(* IEC 61131-3 sources: std_i2980_v2.06_cp053/Source/IMM/ieccontrol/GlobalBaseArchives (part 5) *)

(* ---- FBStart.pu ---- *)
(*
IntermediateCond is optional(only needed for movements with intermediate conditions)
It starts from 1 to and goes up to the maximum intermediate condition
For movements without intermediate conditions it should be 0.

*)

IMPORT_OVER_LISTFILE
 SET_EVENT
, ASSERT
, tsDeviceId
, tMoveIdent
, tsMoveData
, tevStartData
, tevStart

END_IMPORT

FUNCTION_BLOCK FBStart #DUMMY_EDIT_BLOCK

VAR_INPUT
 DeviceId : tsDeviceId (* Device that should be started *);
 MoveDir : tMoveIdent (* Movement direction to start *);
 MoveId : tMoveIdent (* Movement ID to start *);
 IntermediateCond : DINT (* optional: Intermediate condition that should be used for the movement *);
 pbPosReached : REFTO BOOL (* optional: *);
 pMovementData : REFTO tsMoveData (* optional: Reference to the sv_MoveXxx *);
END_VAR

SYSTEM_VAR
 sv_bInitDone : BOOL;
END_VAR

SYSTEM_OBJECT
 evStart : tevStart;
 erAssert : ALARM;
END_OBJECT

VAR
 evStartData : tevStartData;
 dummy : BOOL;
END_VAR
#BEGIN_EDIT_BLOCK
(**************************************** WARNING ********************************************
 *** The KEBA Kemro K2 System including software is not intended for safety control tasks! ***
 ***                       For further information see Comment tab!                        ***
 *********************************************************************************************)

//if the movements are still not registered, gives application programmer code offset and frame offset
dummy := ASSERT(sv_bInitDone, erAssert);

//send start event
evStartData.DeviceId := DeviceId;
evStartData.MoveDir := MoveDir;
evStartData.MoveId := MoveId;
evStartData.IntermediateCond := IntermediateCond;
evStartData.pbPosReached := pbPosReached;
evStartData.pMovementData := pMovementData;
SET_EVENT(evStart,evStartData);

;#END_EDIT_BLOCK END_FUNCTION_BLOCK

#END_OF_IEC_PART

@Puma @IecEditor 6 96 @Pou 25
@@@BEG_Comment@@@
IntermediateCond is optional(only needed for movements with intermediate conditions)
It starts from 1 to and goes up to the maximum intermediate condition
For movements without intermediate conditions it should be 0.

@@@END_Comment@@@

@BEG_Contents

@BEG_Func
@RT(17)FuncTreeContainer
2
@Var @RT(9)SET_EVENT @RT(0) @T @T @DERIVED 0 @F @RT(23)KEBA_STANDARD_PROCEDURE @F
@T
@BEG_Attrib
0 @RT(0) @RT(0)
@END_Attrib
1 1 @F @F @F @F

@Var @RT(6)ASSERT @RT(0) @T @T @DERIVED 0 @F @RT(8)FUNCTION @F
@T
@BEG_Attrib
0 @RT(0) @RT(0)
@END_Attrib
1 1 @F @F @F @F

@END_Func

@BEG_Const
@RT(18)ConstTreeContainer
0
@END_Const

@BEG_Export

@BEG_Kind
@FUNCTION_BLOCK @RT(7)FBStart @STRUCTURED_TEXT
@RT(0) @RT(0) @RT(0)
@END_Kind

@BEG_Dcl
@RT(16)DclTreeContainer
11
@Var @RT(8)DeviceId @RT(0) @T @T @DERIVED 0 @T @T @DT @RT(10)tsDeviceId @RT(0) @T @T @UNKNOWN 0 @F
@F @F
@T
@BEG_Attrib
3 @RT(0) @RT(29)Device that should be started @RT(0)
@END_Attrib
1 1 @F @F @F @F

@Var @RT(7)MoveDir @RT(0) @T @T @DERIVED 0 @T @T @DT @RT(10)tMoveIdent @RT(0) @T @T @UNKNOWN 0 @F
@F @F
@T
@BEG_Attrib
3 @RT(0) @RT(27)Movement direction to start @RT(0)
@END_Attrib
1 1 @F @F @F @F

@Var @RT(6)MoveId @RT(0) @T @T @DERIVED 0 @T @T @DT @RT(10)tMoveIdent @RT(0) @T @T @UNKNOWN 0 @F
@F @F
@T
@BEG_Attrib
3 @RT(0) @RT(20)Movement ID to start @RT(0)
@END_Attrib
1 1 @F @F @F @F

@Var @RT(16)IntermediateCond @RT(0) @T @F @DT @RT(4)DINT @RT(0) @T @T @BASIC 0 @F
@F @F
@T
@BEG_Attrib
3 @RT(0) @RT(69)optional: Intermediate condition that should be used for the movement @RT(0)
@END_Attrib
1 1 @F @F @F @F

@Var @RT(12)pbPosReached @RT(0) @T @T @REFTO 0 @T @DT @RT(4)BOOL @RT(0) @T @T @BASIC 0 @F
@F @F
@T
@BEG_Attrib
3 @RT(0) @RT(9)optional: @RT(0)
@END_Attrib
1 1 @F @F @F @F

@Var @RT(13)pMovementData @RT(0) @T @T @REFTO 0 @F @DERIVED 0 @T @T @DT @RT(10)tsMoveData @RT(0) @T @T @UNKNOWN 0 @F
@F @F
@T
@BEG_Attrib
3 @RT(0) @RT(37)optional: Reference to the sv_MoveXxx @RT(0)
@END_Attrib
1 1 @F @F @F @F

@Var @RT(11)evStartData @RT(0) @T @T @DERIVED 0 @T @T @DT @RT(12)tevStartData @RT(0) @T @T @UNKNOWN 0 @F
@F @F
@T
@BEG_Attrib
3 @RT(0) @RT(0) @RT(0)
@END_Attrib
1 0 @F @F @F @F

@Var @RT(7)evStart @RT(0) @T @T @DERIVED 0 @T @T @DT @RT(8)tevStart @RT(0) @T @T @UNKNOWN 0 @F
@F @F
@T
@BEG_Attrib
3 @RT(0) @RT(0) @RT(0)
@END_Attrib
1 7 @F @F @F @F

@Var @RT(5)dummy @RT(0) @T @F @DT @RT(4)BOOL @RT(0) @T @T @BASIC 0 @F
@F @F
@T
@BEG_Attrib
3 @RT(0) @RT(0) @RT(0)
@END_Attrib
1 0 @F @F @F @F

@Var @RT(12)sv_bInitDone @RT(0) @T @F @DT @RT(4)BOOL @RT(0) @T @T @BASIC 0 @F
@F @F
@T
@BEG_Attrib
3 @RT(0) @RT(0) @RT(0)
@END_Attrib
1 8 @F @F @F @F

@Var @RT(8)erAssert @RT(0) @T @F @DT @RT(5)ALARM @RT(0) @T @T @BASIC 0 @F
@F @F
@T
@BEG_Attrib
3 @RT(0) @RT(0) @RT(0)
@END_Attrib
1 7 @F @F @F @F

@END_Dcl

@END_Export

@BEG_Body
@TL(20)
(**************************************** WARNING ********************************************
 *** The KEBA Kemro K2 System including software is not intended for safety control tasks! ***
 ***                       For further information see Comment tab!                        ***
 *********************************************************************************************)

//if the movements are still not registered, gives application programmer code offset and frame offset
dummy := ASSERT(sv_bInitDone, erAssert);

//send start event
evStartData.DeviceId := DeviceId;
evStartData.MoveDir := MoveDir;
evStartData.MoveId := MoveId;
evStartData.IntermediateCond := IntermediateCond;
evStartData.pbPosReached := pbPosReached;
evStartData.pMovementData := pMovementData;
SET_EVENT(evStart,evStartData);

@END_Body

@END_Contents

(* ---- FBStop.pu ---- *)
IMPORT_OVER_LISTFILE
 ASSERT
, tsDeviceId
, tevStop
, tevStopData

END_IMPORT

FUNCTION_BLOCK FBStop #DUMMY_EDIT_BLOCK

VAR_INPUT
 DeviceId : tsDeviceId;
END_VAR

SYSTEM_VAR
 sv_bInitDone : BOOL;
END_VAR

SYSTEM_OBJECT
 evStop : tevStop;
 erAssert : ALARM;
END_OBJECT

VAR
 evStopData : tevStopData;
 dummy : BOOL;
END_VAR
#BEGIN_EDIT_BLOCK
(**************************************** WARNING ********************************************
 *** The KEBA Kemro K2 System including software is not intended for safety control tasks! ***
 ***                       For further information see Comment tab!                        ***
 *********************************************************************************************)

//if the movements are still not registered, gives application programmer code offset and frame offset
dummy := ASSERT(sv_bInitDone, erAssert);

evStopData.DeviceId := DeviceId;
SET_EVENT(evStop, evStopData);

;#END_EDIT_BLOCK END_FUNCTION_BLOCK

#END_OF_IEC_PART

@Puma @IecEditor 6 10 @Pou 25
@@@BEG_Comment@@@

@@@END_Comment@@@

@BEG_Contents

@BEG_Func
@RT(17)FuncTreeContainer
1
@Var @RT(6)ASSERT @RT(0) @T @T @DERIVED 0 @F @RT(15)FUNCTION : BOOL @F
@T
@BEG_Attrib
0 @RT(0) @RT(0)
@END_Attrib
1 1 @F @F @F @F

@END_Func

@BEG_Const
@RT(18)ConstTreeContainer
0
@END_Const

@BEG_Export

@BEG_Kind
@FUNCTION_BLOCK @RT(6)FBStop @STRUCTURED_TEXT
@RT(0) @RT(0) @RT(0)
@END_Kind

@BEG_Dcl
@RT(16)DclTreeContainer
6
@Var @RT(8)DeviceId @RT(0) @T @T @DERIVED 0 @T @T @DT @RT(10)tsDeviceId @RT(0) @T @T @UNKNOWN 0 @F
@F @F
@T
@BEG_Attrib
3 @RT(0) @RT(0) @RT(0)
@END_Attrib
1 1 @F @F @F @F

@Var @RT(6)evStop @RT(0) @T @T @DERIVED 0 @T @T @DT @RT(7)tevStop @RT(0) @T @T @UNKNOWN 0 @F
@F @F
@T
@BEG_Attrib
3 @RT(0) @RT(0) @RT(0)
@END_Attrib
1 7 @F @F @F @F

@Var @RT(10)evStopData @RT(0) @T @T @DERIVED 0 @T @T @DT @RT(11)tevStopData @RT(0) @T @T @UNKNOWN 0 @F
@F @F
@T
@BEG_Attrib
3 @RT(0) @RT(0) @RT(0)
@END_Attrib
1 0 @F @F @F @F

@Var @RT(8)erAssert @RT(0) @T @F @DT @RT(5)ALARM @RT(0) @T @T @BASIC 0 @F
@F @F
@T
@BEG_Attrib
3 @RT(0) @RT(0) @RT(0)
@END_Attrib
1 7 @F @F @F @F

@Var @RT(5)dummy @RT(0) @T @F @DT @RT(4)BOOL @RT(0) @T @T @BASIC 0 @F
@F @F
@T
@BEG_Attrib
3 @RT(0) @RT(0) @RT(0)
@END_Attrib
1 0 @F @F @F @F

@Var @RT(12)sv_bInitDone @RT(0) @T @F @DT @RT(4)BOOL @RT(0) @T @T @BASIC 0 @F
@F @F
@T
@BEG_Attrib
3 @RT(0) @RT(0) @RT(0)
@END_Attrib
1 8 @F @F @F @F

@END_Dcl

@END_Export

@BEG_Body
@TL(11)
(**************************************** WARNING ********************************************
 *** The KEBA Kemro K2 System including software is not intended for safety control tasks! ***
 ***                       For further information see Comment tab!                        ***
 *********************************************************************************************)

//if the movements are still not registered, gives application programmer code offset and frame offset
dummy := ASSERT(sv_bInitDone, erAssert);

evStopData.DeviceId := DeviceId;
SET_EVENT(evStop, evStopData);

@END_Body

@END_Contents

(* ---- FBStopStartedMovements.pu ---- *)
(*
@h    ! WARNING !
@h    The Kemro K2 system (including software) only meets category B according to EN 954-1,
@h    thus it is not intended for usage in safety-relevant control applications in the field
@h    of personal safety (e.g. emergency stop).
@h    To implement potentially necessary safety-relevant control tasks, always use additional
@h    external safety devices that are intended for the particular purpose, and meet the necessary
@h    functional safety.
@h    For further information see EN 954-1 (EN ISO 13849-1) and/or the K2-x00 user manual, chapter
@h    "CE conformity, directives and standards".
*)

IMPORT_OVER_LISTFILE
 tsStartedMoveData
, FBDebugTrace2
, FBStop

END_IMPORT

FUNCTION_BLOCK FBStopStartedMovements #DUMMY_EDIT_BLOCK

SYSTEM_VAR
 sv_StartedMovements : tsStartedMoveData;
END_VAR

VAR_TEMP
 i : DINT;
END_VAR

VAR
 StartedMovements : tsStartedMoveData;
 fbDebugTrace2 : FBDebugTrace2;
 fbStop : FBStop;
END_VAR
#BEGIN_EDIT_BLOCK
(**************************************** WARNING ********************************************
 *** The KEBA Kemro K2 System including software is not intended for safety control tasks! ***
 ***                       For further information see Comment tab!                        ***
 *********************************************************************************************)

//copy systemvariable to local variable because systemvariable can be changed during executing the code
StartedMovements := sv_StartedMovements;

FOR i := 1 TO StartedMovements.iStartedMovements DO
   //stop all started movements
   fbDebugTrace2(nDeviceState, CONCAT('FBStopStartedMovements.pu stopping device ',
                 DINT_TO_STRING(StartedMovements.MoveData[i].DeviceId.CompId),
                 '/',
                 DINT_TO_STRING(StartedMovements.MoveData[i].DeviceId.IndexId),
                 ' (list entry ',
                 DINT_TO_STRING(i),
                 ' of ',
                 DINT_TO_STRING(StartedMovements.iStartedMovements),
                 ')'));
   fbStop(DeviceId := StartedMovements.MoveData[i].DeviceId);
END_FOR;

;#END_EDIT_BLOCK END_FUNCTION_BLOCK

#END_OF_IEC_PART

@Puma @IecEditor 6 94 @Pou 25
@@@BEG_Comment@@@
@h    ! WARNING !
@h    The Kemro K2 system (including software) only meets category B according to EN 954-1,
@h    thus it is not intended for usage in safety-relevant control applications in the field
@h    of personal safety (e.g. emergency stop).
@h    To implement potentially necessary safety-relevant control tasks, always use additional
@h    external safety devices that are intended for the particular purpose, and meet the necessary
@h    functional safety.
@h    For further information see EN 954-1 (EN ISO 13849-1) and/or the K2-x00 user manual, chapter
@h    "CE conformity, directives and standards".
@@@END_Comment@@@

@BEG_Contents

@BEG_Func
@RT(17)FuncTreeContainer
0
@END_Func

@BEG_Const
@RT(18)ConstTreeContainer
0
@END_Const

@BEG_Export

@BEG_Kind
@FUNCTION_BLOCK @RT(22)FBStopStartedMovements @STRUCTURED_TEXT
@RT(0) @RT(0) @RT(0)
@END_Kind

@BEG_Dcl
@RT(16)DclTreeContainer
5
@Var @RT(19)sv_StartedMovements @RT(0) @T @T @DERIVED 0 @T @T @DT @RT(17)tsStartedMoveData @RT(0) @T @T @UNKNOWN 0 @F
@F @F
@T
@BEG_Attrib
3 @RT(0) @RT(0) @RT(0)
@END_Attrib
1 8 @F @F @F @F

@Var @RT(16)StartedMovements @RT(0) @T @T @DERIVED 0 @T @T @DT @RT(17)tsStartedMoveData @RT(0) @T @T @UNKNOWN 0 @F
@F @F
@T
@BEG_Attrib
3 @RT(0) @RT(0) @RT(0)
@END_Attrib
1 0 @F @F @F @F

@Var @RT(13)fbDebugTrace2 @RT(0) @T @T @DERIVED 0 @F @RT(13)FBDebugTrace2 @F
@T
@BEG_Attrib
3 @RT(0) @RT(0) @RT(0)
@END_Attrib
1 0 @F @F @F @F

@Var @RT(6)fbStop @RT(0) @T @T @DERIVED 0 @T @T @DT @RT(6)FBStop @RT(0) @T @T @UNKNOWN 0 @F
@F @F
@T
@BEG_Attrib
3 @RT(0) @RT(0) @RT(0)
@END_Attrib
1 0 @F @F @F @F

@Var @RT(1)i @RT(0) @T @F @DT @RT(4)DINT @RT(0) @T @T @BASIC 0 @F
@F @F
@T
@BEG_Attrib
3 @RT(0) @RT(0) @RT(0)
@END_Attrib
1 4 @F @F @F @F

@END_Dcl

@END_Export

@BEG_Body
@TL(23)
(**************************************** WARNING ********************************************
 *** The KEBA Kemro K2 System including software is not intended for safety control tasks! ***
 ***                       For further information see Comment tab!                        ***
 *********************************************************************************************)

//copy systemvariable to local variable because systemvariable can be changed during executing the code
StartedMovements := sv_StartedMovements;

FOR i := 1 TO StartedMovements.iStartedMovements DO
   //stop all started movements
   fbDebugTrace2(nDeviceState, CONCAT('FBStopStartedMovements.pu stopping device ',
                 DINT_TO_STRING(StartedMovements.MoveData[i].DeviceId.CompId),
                 '/',
                 DINT_TO_STRING(StartedMovements.MoveData[i].DeviceId.IndexId),
                 ' (list entry ',
                 DINT_TO_STRING(i),
                 ' of ',
                 DINT_TO_STRING(StartedMovements.iStartedMovements),
                 ')'));
   fbStop(DeviceId := StartedMovements.MoveData[i].DeviceId);
END_FOR;

@END_Body

@END_Contents

(* ---- FBTracePendingAlarms.pu ---- *)
(*
This function block traces all pending alarms.
The trace looks like the following example:
1 ExceptionInterpretation1.erCpuFanDefect class: 5 type: 66 SubIDs: 1 1 1 1 - 6338 112 0 0

*)

IMPORT_OVER_LISTFILE
 ALARM_HANDLER
, KSYS_Alarm_Data
, KSYS_Status

END_IMPORT

FUNCTION_BLOCK FBTracePendingAlarms #DUMMY_EDIT_BLOCK

VAR
 abAlarmHandler : ALARM_HANDLER;
 sName : STRING(255);
 AlarmData : KSYS_Alarm_Data;
 Status : KSYS_Status;
 iCounter : DINT;
 dummy : DINT;
END_VAR
#BEGIN_EDIT_BLOCK
(**************************************** WARNING ********************************************
 *** The KEBA Kemro K2 System including software is not intended for safety control tasks! ***
 ***                       For further information see Comment tab!                        ***
 *********************************************************************************************)

iCounter := 1;
dummy := Print('current alarms:');
Status := abAlarmHandler.GetFirstAlarm();
WHILE Status = KSYS_Status_OK DO
   Status := abAlarmHandler.GetAlarmName(AlarmName := sName);
   AlarmData := abAlarmHandler.GetAlarmData();
   dummy := Print('%d %s class: %d type: %d SubIDs: %d %d %d %d - %d %d %d %d', iCounter, sName, AlarmData.Class, AlarmData.Type,
                  AlarmData.SubIDs.SubID1_Used, AlarmData.SubIDs.SubID2_Used, AlarmData.SubIDs.SubID3_Used, AlarmData.SubIDs.SubID4_Used,
                  AlarmData.SubIDs.SubID1, AlarmData.SubIDs.SubID2, AlarmData.SubIDs.SubID3, AlarmData.SubIDs.SubID4);
   Status := abAlarmHandler.GetNextAlarm();
   iCounter := iCounter + 1;
END_WHILE;

;#END_EDIT_BLOCK END_FUNCTION_BLOCK

#END_OF_IEC_PART

@Puma @IecEditor 6 121 @Pou 25
@@@BEG_Comment@@@
This function block traces all pending alarms.
The trace looks like the following example:
1 ExceptionInterpretation1.erCpuFanDefect class: 5 type: 66 SubIDs: 1 1 1 1 - 6338 112 0 0

@@@END_Comment@@@

@BEG_Contents

@BEG_Func
@RT(17)FuncTreeContainer
0
@END_Func

@BEG_Const
@RT(18)ConstTreeContainer
0
@END_Const

@BEG_Export

@BEG_Kind
@FUNCTION_BLOCK @RT(20)FBTracePendingAlarms @STRUCTURED_TEXT
@RT(0) @RT(0) @RT(0)
@END_Kind

@BEG_Dcl
@RT(16)DclTreeContainer
6
@Var @RT(14)abAlarmHandler @RT(0) @T @T @DERIVED 0 @T @T @DT @RT(13)ALARM_HANDLER @RT(0) @T @T @UNKNOWN 0 @F
@F @F
@T
@BEG_Attrib
3 @RT(0) @RT(0) @RT(0)
@END_Attrib
1 0 @F @F @F @F

@Var @RT(5)sName @RT(0) @T @F @DT @RT(11)STRING(255) @RT(0) @T @T @STRING 0 @F @RT(3)255 @F
@F @F
@T
@BEG_Attrib
3 @RT(0) @RT(0) @RT(0)
@END_Attrib
1 0 @F @F @F @F

@Var @RT(9)AlarmData @RT(0) @T @T @DERIVED 0 @T @T @DT @RT(15)KSYS_Alarm_Data @RT(0) @T @T @UNKNOWN 0 @F
@F @F
@T
@BEG_Attrib
3 @RT(0) @RT(0) @RT(0)
@END_Attrib
1 0 @F @F @F @F

@Var @RT(6)Status @RT(0) @T @T @DERIVED 0 @T @T @DT @RT(11)KSYS_Status @RT(0) @T @T @UNKNOWN 0 @F
@F @F
@T
@BEG_Attrib
3 @RT(0) @RT(0) @RT(0)
@END_Attrib
1 0 @F @F @F @F

@Var @RT(8)iCounter @RT(0) @T @F @DT @RT(4)DINT @RT(0) @T @T @BASIC 0 @F
@F @F
@T
@BEG_Attrib
3 @RT(0) @RT(0) @RT(0)
@END_Attrib
1 0 @F @F @F @F

@Var @RT(5)dummy @RT(0) @T @F @DT @RT(4)DINT @RT(0) @T @T @BASIC 0 @F
@F @F
@T
@BEG_Attrib
3 @RT(0) @RT(0) @RT(0)
@END_Attrib
1 0 @F @F @F @F

@END_Dcl

@END_Export

@BEG_Body
@TL(19)
(**************************************** WARNING ********************************************
 *** The KEBA Kemro K2 System including software is not intended for safety control tasks! ***
 ***                       For further information see Comment tab!                        ***
 *********************************************************************************************)

iCounter := 1;
dummy := Print('current alarms:');
Status := abAlarmHandler.GetFirstAlarm();
WHILE Status = KSYS_Status_OK DO
   Status := abAlarmHandler.GetAlarmName(AlarmName := sName);
   AlarmData := abAlarmHandler.GetAlarmData();
   dummy := Print('%d %s class: %d type: %d SubIDs: %d %d %d %d - %d %d %d %d', iCounter, sName, AlarmData.Class, AlarmData.Type,
                  AlarmData.SubIDs.SubID1_Used, AlarmData.SubIDs.SubID2_Used, AlarmData.SubIDs.SubID3_Used, AlarmData.SubIDs.SubID4_Used,
                  AlarmData.SubIDs.SubID1, AlarmData.SubIDs.SubID2, AlarmData.SubIDs.SubID3, AlarmData.SubIDs.SubID4);
   Status := abAlarmHandler.GetNextAlarm();
   iCounter := iCounter + 1;
END_WHILE;

@END_Body

@END_Contents

(* ---- FBUpdateEditorProperties.pu ---- *)
(*
@h    ! WARNING !
@h    The Kemro K2 system (including software) only meets category B according to EN 954-1,
@h    thus it is not intended for usage in safety-relevant control applications in the field
@h    of personal safety (e.g. emergency stop).
@h    To implement potentially necessary safety-relevant control tasks, always use additional
@h    external safety devices that are intended for the particular purpose, and meet the necessary
@h    functional safety.
@h    For further information see EN 954-1 (EN ISO 13849-1) and/or the K2-x00 user manual, chapter
@h    "CE conformity, directives and standards".

The movement duration is updated by ODC after the movement finishes in half - or fullauto cycle.
If the movement duration was not outside the tolerance the editor should not update the properties.
In this case the systemvariable sv_iDurationUpdateInTolerance is increased by ODC.
The according postupdates which react on changes of the duration must check sv_iDurationUpdateInTolerance and
should only trigger the editor update if sv_iDurationUpdateInTolerance is 0 (=duration change outside the tolerance)
*)

FUNCTION_BLOCK FBUpdateEditorProperties #DUMMY_EDIT_BLOCK

SYSTEM_VAR
 sv_iEditorPropertiesChanged : DINT;
 sv_iDurationUpdateInTolerance : DINT;
END_VAR
#BEGIN_EDIT_BLOCK
(**************************************** WARNING ********************************************
 *** The KEBA Kemro K2 System including software is not intended for safety control tasks! ***
 ***                       For further information see Comment tab!                        ***
 *********************************************************************************************)

IF sv_iDurationUpdateInTolerance <> 0 THEN
   //duration was corrected by ABInterpreter (ODC) although it was in tolerance
   //-> don´t trigger update of editor
   //only decrease sv_iDurationUpdateInTolerance
   sv_iDurationUpdateInTolerance := sv_iDurationUpdateInTolerance -1;
ELSE
   //trigger update of editor properties
   sv_iEditorPropertiesChanged := sv_iEditorPropertiesChanged + 1;
END_IF;

;#END_EDIT_BLOCK END_FUNCTION_BLOCK

#END_OF_IEC_PART

@Puma @IecEditor 6 114 @Pou 25
@@@BEG_Comment@@@
@h    ! WARNING !
@h    The Kemro K2 system (including software) only meets category B according to EN 954-1,
@h    thus it is not intended for usage in safety-relevant control applications in the field
@h    of personal safety (e.g. emergency stop).
@h    To implement potentially necessary safety-relevant control tasks, always use additional
@h    external safety devices that are intended for the particular purpose, and meet the necessary
@h    functional safety.
@h    For further information see EN 954-1 (EN ISO 13849-1) and/or the K2-x00 user manual, chapter
@h    "CE conformity, directives and standards".

The movement duration is updated by ODC after the movement finishes in half - or fullauto cycle.
If the movement duration was not outside the tolerance the editor should not update the properties.
In this case the systemvariable sv_iDurationUpdateInTolerance is increased by ODC.
The according postupdates which react on changes of the duration must check sv_iDurationUpdateInTolerance and
should only trigger the editor update if sv_iDurationUpdateInTolerance is 0 (=duration change outside the tolerance)
@@@END_Comment@@@

@BEG_Contents

@BEG_Func
@RT(17)FuncTreeContainer
0
@END_Func

@BEG_Const
@RT(18)ConstTreeContainer
0
@END_Const

@BEG_Export

@BEG_Kind
@FUNCTION_BLOCK @RT(24)FBUpdateEditorProperties @STRUCTURED_TEXT
@RT(0) @RT(0) @RT(0)
@END_Kind

@BEG_Dcl
@RT(16)DclTreeContainer
2
@Var @RT(27)sv_iEditorPropertiesChanged @RT(0) @T @T @RENAMED 0 @T @T @DT @RT(4)DINT @RT(0) @T @T @BASIC 0 @F
@F @F
@T
@BEG_Attrib
3 @RT(0) @RT(0) @RT(0)
@END_Attrib
1 8 @F @F @F @F

@Var @RT(29)sv_iDurationUpdateInTolerance @RT(0) @T @F @DT @RT(4)DINT @RT(0) @T @T @BASIC 0 @F
@F @F
@T
@BEG_Attrib
3 @RT(0) @RT(0) @RT(0)
@END_Attrib
1 8 @F @F @F @F

@END_Dcl

@END_Export

@BEG_Body
@TL(18)
(**************************************** WARNING ********************************************
 *** The KEBA Kemro K2 System including software is not intended for safety control tasks! ***
 ***                       For further information see Comment tab!                        ***
 *********************************************************************************************)

IF sv_iDurationUpdateInTolerance <> 0 THEN
   //duration was corrected by ABInterpreter (ODC) although it was in tolerance
   //-> don´t trigger update of editor
   //only decrease sv_iDurationUpdateInTolerance
   sv_iDurationUpdateInTolerance := sv_iDurationUpdateInTolerance -1;
ELSE
   //trigger update of editor properties
   sv_iEditorPropertiesChanged := sv_iEditorPropertiesChanged + 1;
END_IF;

@END_Body

@END_Contents

(* ---- ABAnalogOutput.pu ---- *)
(*
@h    ! WARNING !
@h    The Kemro K2 system (including software) only meets category B according to EN 954-1,
@h    thus it is not intended for usage in safety-relevant control applications in the field
@h    of personal safety (e.g. emergency stop).
@h    To implement potentially necessary safety-relevant control tasks, always use additional
@h    external safety devices that are intended for the particular purpose, and meet the necessary
@h    functional safety.
@h    For further information see EN 954-1 (EN ISO 13849-1) and/or the K2-x00 user manual, chapter
@h    "CE conformity, directives and standards".

Setvalue linearisation for AnalogOutput with automatic update on change of Lintab SV.

*)

IMPORT_OVER_LISTFILE
 KAPPL_LintabData
, KAPPL_Plastics_Output

END_IMPORT

ALGORITHM_BLOCK ABAnalogOutput #DUMMY_EDIT_BLOCK

SYSTEM_OBJECT
 PU_Task_7 : TASK;
END_OBJECT

VAR
 mpLintab : REFTO KAPPL_LintabData;
 mbReParam : BOOL;
END_VAR

ALGORITHM aInit

VAR_INPUT
 pLintab : REFTO KAPPL_LintabData (* reference to SV with Linearisation Table *);
END_VAR

VAR
 pOldLintab : REFTO KAPPL_LintabData;
END_VAR
#BEGIN_EDIT_BLOCK
(**************************************** WARNING ********************************************
 *** The KEBA Kemro K2 System including software is not intended for safety control tasks! ***
 ***                       For further information see Comment tab!                        ***
 *********************************************************************************************)

IF pLintab <> pOldLintab THEN
   //copy reference
   mpLintab := pLintab;
   mbReParam := TRUE;
   pOldLintab := pLintab;
END_IF;

;#END_EDIT_BLOCK END_ALGORITHM

POSTUPDATE_ALGORITHM pParametersChanged ON PU_Task_7 WITH mpLintab^

#BEGIN_EDIT_BLOCK
(**************************************** WARNING ********************************************
 *** The KEBA Kemro K2 System including software is not intended for safety control tasks! ***
 ***                       For further information see Comment tab!                        ***
 *********************************************************************************************)

mbReParam := TRUE;

;#END_EDIT_BLOCK END_ALGORITHM

(*
Lintab calculation
*)

ALGORITHM aRun

VAR_INPUT
 rSetValue : REAL (* input value *);
END_VAR

VAR_OUTPUT
 rOutput : REAL (* analog output value *);
 bError : BOOL (* error occured *);
 iErrorInfo : DINT (* additional error info *);
END_VAR

VAR
 fbOutput : KAPPL_Plastics_Output;
END_VAR
#BEGIN_EDIT_BLOCK
(**************************************** WARNING ********************************************
 *** The KEBA Kemro K2 System including software is not intended for safety control tasks! ***
 ***                       For further information see Comment tab!                        ***
 *********************************************************************************************)

IF mbReParam THEN
    fbOutput(CycleTime := GET_TASK_INTERVAL(),
             Lintab := mpLintab^,
             Ramps := 999999.9,
             ReParam := TRUE);

    mbReParam := FALSE;
END_IF;

//cyclic part
fbOutput(SetValue := rSetValue,
         ReParam := FALSE);

rOutput := fbOutput.OutputValue;
bError := fbOutput.Error;
iErrorInfo := fbOutput.ErrorInfo;

;#END_EDIT_BLOCK END_ALGORITHM

END_ALGORITHM_BLOCK

#END_OF_IEC_PART

@Puma @IecEditor 6 10 @Pou 25
@@@BEG_Comment@@@
@h    ! WARNING !
@h    The Kemro K2 system (including software) only meets category B according to EN 954-1,
@h    thus it is not intended for usage in safety-relevant control applications in the field
@h    of personal safety (e.g. emergency stop).
@h    To implement potentially necessary safety-relevant control tasks, always use additional
@h    external safety devices that are intended for the particular purpose, and meet the necessary
@h    functional safety.
@h    For further information see EN 954-1 (EN ISO 13849-1) and/or the K2-x00 user manual, chapter
@h    "CE conformity, directives and standards".

Setvalue linearisation for AnalogOutput with automatic update on change of Lintab SV.

@@@END_Comment@@@

@BEG_Contents

@BEG_Func
@RT(17)FuncTreeContainer
0
@END_Func

@BEG_Const
@RT(18)ConstTreeContainer
0
@END_Const

@BEG_Export

@BEG_Kind
@ALGORITHM_BLOCK @RT(14)ABAnalogOutput @STRUCTURED_TEXT
@RT(0) @RT(0) @RT(0)
@END_Kind

@BEG_Dcl
@RT(16)DclTreeContainer
3
@Var @RT(9)PU_Task_7 @RT(0) @T @T @RENAMED 0 @T @T @DT @RT(4)TASK @RT(0) @T @T @BASIC 0 @F
@F @F
@T
@BEG_Attrib
3 @RT(0) @RT(0) @RT(0)
@END_Attrib
1 7 @F @F @F @F

@Var @RT(8)mpLintab @RT(0) @T @T @REFTO 0 @F @DERIVED 0 @T @T @DT @RT(16)KAPPL_LintabData @RT(0) @T @T @UNKNOWN 0 @F
@F @F
@T
@BEG_Attrib
3 @RT(0) @RT(0) @RT(0)
@END_Attrib
1 0 @F @F @F @F

@Var @RT(9)mbReParam @RT(0) @T @F @DT @RT(4)BOOL @RT(0) @T @T @BASIC 0 @F
@F @F
@T
@BEG_Attrib
3 @RT(0) @RT(0) @RT(0)
@END_Attrib
1 0 @F @F @F @F

@END_Dcl

@END_Export

@BEG_Body

3

@BEG_Export

@BEG_Algo
@ALGORITHM @RT(5)aInit @STRUCTURED_TEXT
@RT(0) @RT(0) @RT(0) @F @F
@END_Algo

@BEG_Dcl
@RT(16)DclTreeContainer
2
@Var @RT(7)pLintab @RT(0) @T @T @REFTO 0 @F @DERIVED 0 @T @T @DT @RT(16)KAPPL_LintabData @RT(0) @T @T @UNKNOWN 0 @F
@F @F
@T
@BEG_Attrib
3 @RT(0) @RT(40)reference to SV with Linearisation Table @RT(0)
@END_Attrib
1 1 @F @F @F @F

@Var @RT(10)pOldLintab @RT(0) @T @T @REFTO 0 @F @DERIVED 0 @T @T @DT @RT(16)KAPPL_LintabData @RT(0) @T @T @UNKNOWN 0 @F
@F @F
@T
@BEG_Attrib
3 @RT(0) @RT(0) @RT(0)
@END_Attrib
1 0 @F @F @F @F

@END_Dcl

@END_Export

@BEG_Export

@BEG_Algo
@POSTUPDATE_ALGORITHM @RT(18)pParametersChanged @STRUCTURED_TEXT
@RT(0) @RT(9)mpLintab^ @RT(9)PU_Task_7 @F @F
@END_Algo

@BEG_Dcl
@RT(16)DclTreeContainer
0
@END_Dcl

@END_Export

@BEG_Export

@BEG_Algo
@ALGORITHM @RT(4)aRun @STRUCTURED_TEXT
@RT(0) @RT(0) @RT(0) @F @F
@END_Algo

@BEG_Dcl
@RT(16)DclTreeContainer
5
@Var @RT(9)rSetValue @RT(0) @T @F @DT @RT(4)REAL @RT(0) @T @T @BASIC 0 @F
@F @F
@T
@BEG_Attrib
3 @RT(0) @RT(11)input value @RT(0)
@END_Attrib
1 1 @F @F @F @F

@Var @RT(7)rOutput @RT(0) @T @F @DT @RT(4)REAL @RT(0) @T @T @BASIC 0 @F
@F @F
@T
@BEG_Attrib
3 @RT(0) @RT(19)analog output value @RT(0)
@END_Attrib
1 3 @F @F @F @F

@Var @RT(6)bError @RT(0) @T @F @DT @RT(4)BOOL @RT(0) @T @T @BASIC 0 @F
@F @F
@T
@BEG_Attrib
3 @RT(0) @RT(13)error occured @RT(0)
@END_Attrib
1 3 @F @F @F @F

@Var @RT(10)iErrorInfo @RT(0) @T @F @DT @RT(4)DINT @RT(0) @T @T @BASIC 0 @F
@F @F
@T
@BEG_Attrib
3 @RT(0) @RT(21)additional error info @RT(0)
@END_Attrib
1 3 @F @F @F @F

@Var @RT(8)fbOutput @RT(0) @T @T @DERIVED 0 @T @T @DT @RT(21)KAPPL_Plastics_Output @RT(0) @T @T @UNKNOWN 0 @F
@F @F
@T
@BEG_Attrib
3 @RT(0) @RT(0) @RT(0)
@END_Attrib
1 0 @F @F @F @F

@END_Dcl

@END_Export

@BEG_Body
@TL(12)
(**************************************** WARNING ********************************************
 *** The KEBA Kemro K2 System including software is not intended for safety control tasks! ***
 ***                       For further information see Comment tab!                        ***
 *********************************************************************************************)

IF pLintab <> pOldLintab THEN
   //copy reference
   mpLintab := pLintab;
   mbReParam := TRUE;
   pOldLintab := pLintab;
END_IF;

@END_Body

@@@BEG_Comment@@@
@TL(0)

@@@END_Comment@@@

@BEG_Body
@TL(7)
(**************************************** WARNING ********************************************
 *** The KEBA Kemro K2 System including software is not intended for safety control tasks! ***
 ***                       For further information see Comment tab!                        ***
 *********************************************************************************************)

mbReParam := TRUE;

@END_Body

@@@BEG_Comment@@@
@TL(0)

@@@END_Comment@@@

@BEG_Body
@TL(24)
(**************************************** WARNING ********************************************
 *** The KEBA Kemro K2 System including software is not intended for safety control tasks! ***
 ***                       For further information see Comment tab!                        ***
 *********************************************************************************************)

IF mbReParam THEN
    fbOutput(CycleTime := GET_TASK_INTERVAL(),
             Lintab := mpLintab^,
             Ramps := 999999.9,
             ReParam := TRUE);

    mbReParam := FALSE;
END_IF;

//cyclic part
fbOutput(SetValue := rSetValue,
         ReParam := FALSE);

rOutput := fbOutput.OutputValue;
bError := fbOutput.Error;
iErrorInfo := fbOutput.ErrorInfo;

@END_Body

@@@BEG_Comment@@@
@TL(1)
Lintab calculation
@@@END_Comment@@@
@END_Body

@END_Contents

(* ---- ABAutoCalibRedoListener.pu ---- *)
(*
@h    ! WARNING !
@h    The Kemro K2 system (including software) only meets category B according to EN 954-1,
@h    thus it is not intended for usage in safety-relevant control applications in the field
@h    of personal safety (e.g. emergency stop).
@h    To implement potentially necessary safety-relevant control tasks, always use additional
@h    external safety devices that are intended for the particular purpose, and meet the necessary
@h    functional safety.
@h    For further information see EN 954-1 (EN ISO 13849-1) and/or the K2-x00 user manual, chapter
@h    "CE conformity, directives and standards".

wait for a change in the sv_CalibState bRedo or Status fields
If bRedo is set check for Setup mode then send a evRedoStart event
if Status changes away from tnCalibState_Running the bRedo flag is reset
*)

IMPORT_OVER_LISTFILE
 SET_ALARM
, tsCalibMovement
, tevRedoEvent
, tnOperationMode
, tevRedoEventData

END_IMPORT

ALGORITHM_BLOCK ABAutoCalibRedoListener #DUMMY_EDIT_BLOCK

SYSTEM_VAR
 sv_CalibState : tsCalibMovement;
 sv_OperationMode : tnOperationMode;
END_VAR

SYSTEM_OBJECT
 PU_Task_7 : TASK;
 evRedoStart : tevRedoEvent;
 erSetupModeRequiredForCalib : ALARM;
END_OBJECT

(*
@h    ! WARNING !
@h    The Kemro K2 system (including software) only meets category B according to EN 954-1,
@h    thus it is not intended for usage in safety-relevant control applications in the field
@h    of personal safety (e.g. emergency stop).
@h    To implement potentially necessary safety-relevant control tasks, always use additional
@h    external safety devices that are intended for the particular purpose, and meet the necessary
@h    functional safety.
@h    For further information see EN 954-1 (EN ISO 13849-1) and/or the K2-x00 user manual, chapter
@h    "CE conformity, directives and standards".

sets a evRedoStart event, which notifies the autocalibration FU to start this calibration movement
*)

POSTUPDATE_ALGORITHM pUpdateRedo ON PU_Task_7 WITH sv_CalibState.bRedo

VAR_TEMP
 RedoStartData : tevRedoEventData;
END_VAR
#BEGIN_EDIT_BLOCK
(**************************************** WARNING ********************************************
 *** The KEBA Kemro K2 System including software is not intended for safety control tasks! ***
 ***                       For further information see Comment tab!                        ***
 *********************************************************************************************)

IF sv_CalibState.bRedo THEN
    IF sv_OperationMode <> nSetup THEN
       SET_ALARM(erSetupModeRequiredForCalib);
       sv_CalibState.bRedo := FALSE;
       RETURN;
    END_IF;
    RedoStartData.pMovement := @sv_CalibState;
    SET_EVENT(evRedoStart, RedoStartData);
END_IF;

;#END_EDIT_BLOCK END_ALGORITHM

(*
@h    ! WARNING !
@h    The Kemro K2 system (including software) only meets category B according to EN 954-1,
@h    thus it is not intended for usage in safety-relevant control applications in the field
@h    of personal safety (e.g. emergency stop).
@h    To implement potentially necessary safety-relevant control tasks, always use additional
@h    external safety devices that are intended for the particular purpose, and meet the necessary
@h    functional safety.
@h    For further information see EN 954-1 (EN ISO 13849-1) and/or the K2-x00 user manual, chapter
@h    "CE conformity, directives and standards".

sets a evRedoStart event, which notifies the autocalibration FU to start this calibration movement
*)

POSTUPDATE_ALGORITHM pUpdateStatus ON PU_Task_7 WITH sv_CalibState.Status

#BEGIN_EDIT_BLOCK
(**************************************** WARNING ********************************************
 *** The KEBA Kemro K2 System including software is not intended for safety control tasks! ***
 ***                       For further information see Comment tab!                        ***
 *********************************************************************************************)

(* reset bRedo flag, when calibration is finished or aborted *)
IF sv_CalibState.Status <> tnCalibState_Running AND sv_CalibState.bRedo THEN
    sv_CalibState.bRedo := FALSE;
END_IF;

;#END_EDIT_BLOCK END_ALGORITHM

END_ALGORITHM_BLOCK

#END_OF_IEC_PART

@Puma @IecEditor 6 30 @Pou 25
@@@BEG_Comment@@@
@h    ! WARNING !
@h    The Kemro K2 system (including software) only meets category B according to EN 954-1,
@h    thus it is not intended for usage in safety-relevant control applications in the field
@h    of personal safety (e.g. emergency stop).
@h    To implement potentially necessary safety-relevant control tasks, always use additional
@h    external safety devices that are intended for the particular purpose, and meet the necessary
@h    functional safety.
@h    For further information see EN 954-1 (EN ISO 13849-1) and/or the K2-x00 user manual, chapter
@h    "CE conformity, directives and standards".

wait for a change in the sv_CalibState bRedo or Status fields
If bRedo is set check for Setup mode then send a evRedoStart event
if Status changes away from tnCalibState_Running the bRedo flag is reset
@@@END_Comment@@@

@BEG_Contents

@BEG_Func
@RT(17)FuncTreeContainer
1
@Var @RT(9)SET_ALARM @RT(0) @T @T @DERIVED 0 @F @RT(23)KEBA_STANDARD_PROCEDURE @F
@T
@BEG_Attrib
0 @RT(0) @RT(0)
@END_Attrib
1 1 @F @F @F @F

@END_Func

@BEG_Const
@RT(18)ConstTreeContainer
0
@END_Const

@BEG_Export

@BEG_Kind
@ALGORITHM_BLOCK @RT(23)ABAutoCalibRedoListener @STRUCTURED_TEXT
@RT(0) @RT(0) @RT(0)
@END_Kind

@BEG_Dcl
@RT(16)DclTreeContainer
5
@Var @RT(13)sv_CalibState @RT(0) @T @T @DERIVED 0 @T @T @DT @RT(15)tsCalibMovement @RT(0) @T @T @UNKNOWN 0 @F
@F @F
@T
@BEG_Attrib
3 @RT(0) @RT(0) @RT(0)
@END_Attrib
1 8 @F @F @F @F

@Var @RT(9)PU_Task_7 @RT(0) @T @T @RENAMED 0 @T @T @DT @RT(4)TASK @RT(0) @T @T @BASIC 0 @F
@F @F
@T
@BEG_Attrib
3 @RT(0) @RT(0) @RT(0)
@END_Attrib
1 7 @F @F @F @F

@Var @RT(11)evRedoStart @RT(0) @T @T @RENAMED 0 @T @T @DT @RT(12)tevRedoEvent @RT(0) @T @T @UNKNOWN 0 @F
@F @F
@T
@BEG_Attrib
3 @RT(0) @RT(0) @RT(0)
@END_Attrib
1 7 @F @F @F @F

@Var @RT(27)erSetupModeRequiredForCalib @RT(0) @T @T @RENAMED 0 @T @T @DT @RT(5)ALARM @RT(0) @T @T @BASIC 0 @F
@F @F
@T
@BEG_Attrib
3 @RT(0) @RT(0) @RT(0)
@END_Attrib
1 7 @F @F @F @F

@Var @RT(16)sv_OperationMode @RT(0) @T @T @RENAMED 0 @T @T @DT @RT(15)tnOperationMode @RT(0) @T @T @UNKNOWN 0 @F
@F @F
@T
@BEG_Attrib
3 @RT(0) @RT(0) @RT(0)
@END_Attrib
1 8 @F @F @F @F

@END_Dcl

@END_Export

@BEG_Body

2

@BEG_Export

@BEG_Algo
@POSTUPDATE_ALGORITHM @RT(11)pUpdateRedo @STRUCTURED_TEXT
@RT(0) @RT(19)sv_CalibState.bRedo @RT(9)PU_Task_7 @F @F
@END_Algo

@BEG_Dcl
@RT(16)DclTreeContainer
1
@Var @RT(13)RedoStartData @RT(0) @T @T @DERIVED 0 @T @T @DT @RT(16)tevRedoEventData @RT(0) @T @T @UNKNOWN 0 @F
@F @F
@T
@BEG_Attrib
3 @RT(0) @RT(0) @RT(0)
@END_Attrib
1 4 @F @F @F @F

@END_Dcl

@END_Export

@BEG_Export

@BEG_Algo
@POSTUPDATE_ALGORITHM @RT(13)pUpdateStatus @STRUCTURED_TEXT
@RT(0) @RT(20)sv_CalibState.Status @RT(9)PU_Task_7 @F @F
@END_Algo

@BEG_Dcl
@RT(16)DclTreeContainer
0
@END_Dcl

@END_Export

@BEG_Body
@TL(15)
(**************************************** WARNING ********************************************
 *** The KEBA Kemro K2 System including software is not intended for safety control tasks! ***
 ***                       For further information see Comment tab!                        ***
 *********************************************************************************************)

IF sv_CalibState.bRedo THEN
    IF sv_OperationMode <> nSetup THEN
       SET_ALARM(erSetupModeRequiredForCalib);
       sv_CalibState.bRedo := FALSE;
       RETURN;
    END_IF;
    RedoStartData.pMovement := @sv_CalibState;
    SET_EVENT(evRedoStart, RedoStartData);
END_IF;

@END_Body

@@@BEG_Comment@@@
@TL(11)
@h    ! WARNING !
@h    The Kemro K2 system (including software) only meets category B according to EN 954-1,
@h    thus it is not intended for usage in safety-relevant control applications in the field
@h    of personal safety (e.g. emergency stop).
@h    To implement potentially necessary safety-relevant control tasks, always use additional
@h    external safety devices that are intended for the particular purpose, and meet the necessary
@h    functional safety.
@h    For further information see EN 954-1 (EN ISO 13849-1) and/or the K2-x00 user manual, chapter
@h    "CE conformity, directives and standards".

sets a evRedoStart event, which notifies the autocalibration FU to start this calibration movement
@@@END_Comment@@@

@BEG_Body
@TL(10)
(**************************************** WARNING ********************************************
 *** The KEBA Kemro K2 System including software is not intended for safety control tasks! ***
 ***                       For further information see Comment tab!                        ***
 *********************************************************************************************)

(* reset bRedo flag, when calibration is finished or aborted *)
IF sv_CalibState.Status <> tnCalibState_Running AND sv_CalibState.bRedo THEN
    sv_CalibState.bRedo := FALSE;
END_IF;

@END_Body

@@@BEG_Comment@@@
@TL(11)
@h    ! WARNING !
@h    The Kemro K2 system (including software) only meets category B according to EN 954-1,
@h    thus it is not intended for usage in safety-relevant control applications in the field
@h    of personal safety (e.g. emergency stop).
@h    To implement potentially necessary safety-relevant control tasks, always use additional
@h    external safety devices that are intended for the particular purpose, and meet the necessary
@h    functional safety.
@h    For further information see EN 954-1 (EN ISO 13849-1) and/or the K2-x00 user manual, chapter
@h    "CE conformity, directives and standards".

sets a evRedoStart event, which notifies the autocalibration FU to start this calibration movement
@@@END_Comment@@@
@END_Body

@END_Contents

(* ---- ABAutoIdentRedoListener.pu ---- *)
IMPORT_OVER_LISTFILE
 SET_ALARM
, SET_EVENT
, nSetup
, tnCalibState_Running
, tnOperationMode
, tsIdentMovement
, tsIdentSpeedMovement
, tevRedoIdentEvent
, tevRedoIdentSpeedEvent
, tevRedoIdentEventData
, tevRedoIdentSpeedEventData

END_IMPORT

ALGORITHM_BLOCK ABAutoIdentRedoListener #DUMMY_EDIT_BLOCK

SYSTEM_VAR
 sv_OperationMode : tnOperationMode;
 sv_IdentState : tsIdentMovement;
 sv_IdentMaxSpeedState : tsIdentSpeedMovement;
 sv_IdentMinSpeedState : tsIdentSpeedMovement;
END_VAR

SYSTEM_OBJECT
 PU_Task_7 : TASK;
 erSetupModeRequiredForCalib : ALARM;
 evRedoIdentStart : tevRedoIdentEvent;
 evRedoIdentMaxSpeedStart : tevRedoIdentSpeedEvent;
 evRedoIdentMinSpeedStart : tevRedoIdentSpeedEvent;
END_OBJECT

(*
@h    ! WARNING !
@h    The Kemro K2 system (including software) only meets category B according to EN 954-1,
@h    thus it is not intended for usage in safety-relevant control applications in the field
@h    of personal safety (e.g. emergency stop).
@h    To implement potentially necessary safety-relevant control tasks, always use additional
@h    external safety devices that are intended for the particular purpose, and meet the necessary
@h    functional safety.
@h    For further information see EN 954-1 (EN ISO 13849-1) and/or the K2-x00 user manual, chapter
@h    "CE conformity, directives and standards".

sets a evRedoStart event, which notifies the autocalibration FU to start this calibration movement
*)

POSTUPDATE_ALGORITHM pUpdateRedo ON PU_Task_7 WITH sv_IdentState.bRedo

VAR_TEMP
 RedoStartData : tevRedoIdentEventData;
END_VAR
#BEGIN_EDIT_BLOCK
(**************************************** WARNING ********************************************
 *** The KEBA Kemro K2 System including software is not intended for safety control tasks! ***
 ***                       For further information see Comment tab!                        ***
 *********************************************************************************************)

IF sv_IdentState.bRedo THEN
    IF sv_OperationMode <> nSetup THEN
       SET_ALARM(erSetupModeRequiredForCalib);
       sv_IdentState.bRedo := FALSE;
       RETURN;
    END_IF;
    RedoStartData.pMovement := @sv_IdentState;
    SET_EVENT(evRedoIdentStart, RedoStartData);
END_IF;

;#END_EDIT_BLOCK END_ALGORITHM

(*
@h    ! WARNING !
@h    The Kemro K2 system (including software) only meets category B according to EN 954-1,
@h    thus it is not intended for usage in safety-relevant control applications in the field
@h    of personal safety (e.g. emergency stop).
@h    To implement potentially necessary safety-relevant control tasks, always use additional
@h    external safety devices that are intended for the particular purpose, and meet the necessary
@h    functional safety.
@h    For further information see EN 954-1 (EN ISO 13849-1) and/or the K2-x00 user manual, chapter
@h    "CE conformity, directives and standards".

sets a evRedoStart event, which notifies the autocalibration FU to start this calibration movement
*)

POSTUPDATE_ALGORITHM pUpdateStatus ON PU_Task_7 WITH sv_IdentState.Status

#BEGIN_EDIT_BLOCK
(**************************************** WARNING ********************************************
 *** The KEBA Kemro K2 System including software is not intended for safety control tasks! ***
 ***                       For further information see Comment tab!                        ***
 *********************************************************************************************)

(* reset bRedo flag, when calibration is finished or aborted *)
IF sv_IdentState.Status <> tnCalibState_Running AND sv_IdentState.bRedo THEN
    sv_IdentState.bRedo := FALSE;
END_IF;

;#END_EDIT_BLOCK END_ALGORITHM

(*
@h    ! WARNING !
@h    The Kemro K2 system (including software) only meets category B according to EN 954-1,
@h    thus it is not intended for usage in safety-relevant control applications in the field
@h    of personal safety (e.g. emergency stop).
@h    To implement potentially necessary safety-relevant control tasks, always use additional
@h    external safety devices that are intended for the particular purpose, and meet the necessary
@h    functional safety.
@h    For further information see EN 954-1 (EN ISO 13849-1) and/or the K2-x00 user manual, chapter
@h    "CE conformity, directives and standards".

sets a evRedoStart event, which notifies the autocalibration FU to start this calibration movement
*)

POSTUPDATE_ALGORITHM pUpdateMaxRedo ON PU_Task_7 WITH sv_IdentMaxSpeedState.bRedo

VAR_TEMP
 RedoStartData : tevRedoIdentSpeedEventData;
END_VAR
#BEGIN_EDIT_BLOCK
(**************************************** WARNING ********************************************
 *** The KEBA Kemro K2 System including software is not intended for safety control tasks! ***
 ***                       For further information see Comment tab!                        ***
 *********************************************************************************************)

IF sv_IdentMaxSpeedState.bRedo THEN
    IF sv_OperationMode <> nSetup THEN
       SET_ALARM(erSetupModeRequiredForCalib);
       sv_IdentMaxSpeedState.bRedo := FALSE;
       RETURN;
    END_IF;
    RedoStartData.pMovement := @sv_IdentMaxSpeedState;
    SET_EVENT(evRedoIdentMaxSpeedStart, RedoStartData);
END_IF;

;#END_EDIT_BLOCK END_ALGORITHM

(*
@h    ! WARNING !
@h    The Kemro K2 system (including software) only meets category B according to EN 954-1,
@h    thus it is not intended for usage in safety-relevant control applications in the field
@h    of personal safety (e.g. emergency stop).
@h    To implement potentially necessary safety-relevant control tasks, always use additional
@h    external safety devices that are intended for the particular purpose, and meet the necessary
@h    functional safety.
@h    For further information see EN 954-1 (EN ISO 13849-1) and/or the K2-x00 user manual, chapter
@h    "CE conformity, directives and standards".

sets a evRedoStart event, which notifies the autocalibration FU to start this calibration movement
*)

POSTUPDATE_ALGORITHM pUpdateMaxStatus ON PU_Task_7 WITH sv_IdentMaxSpeedState.Status

#BEGIN_EDIT_BLOCK
(**************************************** WARNING ********************************************
 *** The KEBA Kemro K2 System including software is not intended for safety control tasks! ***
 ***                       For further information see Comment tab!                        ***
 *********************************************************************************************)

(* reset bRedo flag, when calibration is finished or aborted *)
IF sv_IdentMaxSpeedState.Status <> tnCalibState_Running AND sv_IdentMaxSpeedState.bRedo THEN
    sv_IdentMaxSpeedState.bRedo := FALSE;
END_IF;

;#END_EDIT_BLOCK END_ALGORITHM

(*
@h    ! WARNING !
@h    The Kemro K2 system (including software) only meets category B according to EN 954-1,
@h    thus it is not intended for usage in safety-relevant control applications in the field
@h    of personal safety (e.g. emergency stop).
@h    To implement potentially necessary safety-relevant control tasks, always use additional
@h    external safety devices that are intended for the particular purpose, and meet the necessary
@h    functional safety.
@h    For further information see EN 954-1 (EN ISO 13849-1) and/or the K2-x00 user manual, chapter
@h    "CE conformity, directives and standards".

sets a evRedoStart event, which notifies the autocalibration FU to start this calibration movement
*)

POSTUPDATE_ALGORITHM pUpdateMinRedo ON PU_Task_7 WITH sv_IdentMinSpeedState.bRedo

VAR_TEMP
 RedoStartData : tevRedoIdentSpeedEventData;
END_VAR
#BEGIN_EDIT_BLOCK
(**************************************** WARNING ********************************************
 *** The KEBA Kemro K2 System including software is not intended for safety control tasks! ***
 ***                       For further information see Comment tab!                        ***
 *********************************************************************************************)

IF sv_IdentMinSpeedState.bRedo THEN
    IF sv_OperationMode <> nSetup THEN
       SET_ALARM(erSetupModeRequiredForCalib);
       sv_IdentMinSpeedState.bRedo := FALSE;
       RETURN;
    END_IF;
    RedoStartData.pMovement := @sv_IdentMinSpeedState;
    SET_EVENT(evRedoIdentMinSpeedStart, RedoStartData);
END_IF;

;#END_EDIT_BLOCK END_ALGORITHM

(*
@h    ! WARNING !
@h    The Kemro K2 system (including software) only meets category B according to EN 954-1,
@h    thus it is not intended for usage in safety-relevant control applications in the field
@h    of personal safety (e.g. emergency stop).
@h    To implement potentially necessary safety-relevant control tasks, always use additional
@h    external safety devices that are intended for the particular purpose, and meet the necessary
@h    functional safety.
@h    For further information see EN 954-1 (EN ISO 13849-1) and/or the K2-x00 user manual, chapter
@h    "CE conformity, directives and standards".

sets a evRedoStart event, which notifies the autocalibration FU to start this calibration movement
*)

POSTUPDATE_ALGORITHM pUpdateMinStatus ON PU_Task_7 WITH sv_IdentMinSpeedState.Status

#BEGIN_EDIT_BLOCK
(**************************************** WARNING ********************************************
 *** The KEBA Kemro K2 System including software is not intended for safety control tasks! ***
 ***                       For further information see Comment tab!                        ***
 *********************************************************************************************)

(* reset bRedo flag, when calibration is finished or aborted *)
IF sv_IdentMinSpeedState.Status <> tnCalibState_Running AND sv_IdentMinSpeedState.bRedo THEN
    sv_IdentMinSpeedState.bRedo := FALSE;
END_IF;

;#END_EDIT_BLOCK END_ALGORITHM

END_ALGORITHM_BLOCK

#END_OF_IEC_PART

@Puma @IecEditor 6 152 @Pou 25
@@@BEG_Comment@@@

@@@END_Comment@@@

@BEG_Contents

@BEG_Func
@RT(17)FuncTreeContainer
2
@Var @RT(9)SET_ALARM @RT(0) @T @T @DERIVED 0 @F @RT(23)KEBA_STANDARD_PROCEDURE @F
@T
@BEG_Attrib
0 @RT(0) @RT(0)
@END_Attrib
1 1 @F @F @F @F

@Var @RT(9)SET_EVENT @RT(0) @T @T @DERIVED 0 @F @RT(23)KEBA_STANDARD_PROCEDURE @F
@T
@BEG_Attrib
0 @RT(0) @RT(0)
@END_Attrib
1 1 @F @F @F @F

@END_Func

@BEG_Const
@RT(18)ConstTreeContainer
2
@Var @RT(6)nSetup @RT(0) @T @T @DERIVED 0 @F @RT(15)tnOperationMode @F
@T
@BEG_Attrib
0 @RT(1)0 @RT(36)Setup mode only for service engineer
@END_Attrib
1 1 @F @F @F @F

@Var @RT(20)tnCalibState_Running @RT(0) @T @T @DERIVED 0 @F @RT(12)tnCalibState @F
@T
@BEG_Attrib
0 @RT(1)1 @RT(23)calibration in progress
@END_Attrib
1 1 @F @F @F @F

@END_Const

@BEG_Export

@BEG_Kind
@ALGORITHM_BLOCK @RT(23)ABAutoIdentRedoListener @STRUCTURED_TEXT
@RT(0) @RT(0) @RT(0)
@END_Kind

@BEG_Dcl
@RT(16)DclTreeContainer
9
@Var @RT(16)sv_OperationMode @RT(0) @T @T @DERIVED 0 @T @T @DT @RT(15)tnOperationMode @RT(0) @T @T @UNKNOWN 0 @F
@F @F
@T
@BEG_Attrib
3 @RT(0) @RT(0) @RT(0)
@END_Attrib
1 8 @F @F @F @F

@Var @RT(13)sv_IdentState @RT(0) @T @T @DERIVED 0 @T @T @DT @RT(15)tsIdentMovement @RT(0) @T @T @UNKNOWN 0 @F
@F @F
@T
@BEG_Attrib
3 @RT(0) @RT(0) @RT(0)
@END_Attrib
1 8 @F @F @F @F

@Var @RT(21)sv_IdentMaxSpeedState @RT(0) @T @T @DERIVED 0 @T @T @DT @RT(20)tsIdentSpeedMovement @RT(0) @T @T @UNKNOWN 0 @F
@F @F
@T
@BEG_Attrib
3 @RT(0) @RT(0) @RT(0)
@END_Attrib
1 8 @F @F @F @F

@Var @RT(21)sv_IdentMinSpeedState @RT(0) @T @T @DERIVED 0 @T @T @DT @RT(20)tsIdentSpeedMovement @RT(0) @T @T @UNKNOWN 0 @F
@F @F
@T
@BEG_Attrib
3 @RT(0) @RT(0) @RT(0)
@END_Attrib
1 8 @F @F @F @F

@Var @RT(9)PU_Task_7 @RT(0) @T @F @DT @RT(4)TASK @RT(0) @T @T @BASIC 0 @F
@F @F
@T
@BEG_Attrib
3 @RT(0) @RT(0) @RT(0)
@END_Attrib
1 7 @F @F @F @F

@Var @RT(27)erSetupModeRequiredForCalib @RT(0) @T @F @DT @RT(5)ALARM @RT(0) @T @T @BASIC 0 @F
@F @F
@T
@BEG_Attrib
3 @RT(0) @RT(0) @RT(0)
@END_Attrib
1 7 @F @F @F @F

@Var @RT(16)evRedoIdentStart @RT(0) @T @T @DERIVED 0 @T @T @DT @RT(17)tevRedoIdentEvent @RT(0) @T @T @UNKNOWN 0 @F
@F @F
@T
@BEG_Attrib
3 @RT(0) @RT(0) @RT(0)
@END_Attrib
1 7 @F @F @F @F

@Var @RT(24)evRedoIdentMaxSpeedStart @RT(0) @T @T @DERIVED 0 @T @T @DT @RT(22)tevRedoIdentSpeedEvent @RT(0) @T @T @UNKNOWN 0 @F
@F @F
@T
@BEG_Attrib
3 @RT(0) @RT(0) @RT(0)
@END_Attrib
1 7 @F @F @F @F

@Var @RT(24)evRedoIdentMinSpeedStart @RT(0) @T @T @DERIVED 0 @T @T @DT @RT(22)tevRedoIdentSpeedEvent @RT(0) @T @T @UNKNOWN 0 @F
@F @F
@T
@BEG_Attrib
3 @RT(0) @RT(0) @RT(0)
@END_Attrib
1 7 @F @F @F @F

@END_Dcl

@END_Export

@BEG_Body

6

@BEG_Export

@BEG_Algo
@POSTUPDATE_ALGORITHM @RT(11)pUpdateRedo @STRUCTURED_TEXT
@RT(0) @RT(19)sv_IdentState.bRedo @RT(9)PU_Task_7 @F @F
@END_Algo

@BEG_Dcl
@RT(16)DclTreeContainer
1
@Var @RT(13)RedoStartData @RT(0) @T @T @DERIVED 0 @T @T @DT @RT(21)tevRedoIdentEventData @RT(0) @T @T @UNKNOWN 0 @F
@F @F
@T
@BEG_Attrib
3 @RT(0) @RT(0) @RT(0)
@END_Attrib
1 4 @F @F @F @F

@END_Dcl

@END_Export

@BEG_Export

@BEG_Algo
@POSTUPDATE_ALGORITHM @RT(13)pUpdateStatus @STRUCTURED_TEXT
@RT(0) @RT(20)sv_IdentState.Status @RT(9)PU_Task_7 @F @F
@END_Algo

@BEG_Dcl
@RT(16)DclTreeContainer
0
@END_Dcl

@END_Export

@BEG_Export

@BEG_Algo
@POSTUPDATE_ALGORITHM @RT(14)pUpdateMaxRedo @STRUCTURED_TEXT
@RT(0) @RT(27)sv_IdentMaxSpeedState.bRedo @RT(9)PU_Task_7 @F @F
@END_Algo

@BEG_Dcl
@RT(16)DclTreeContainer
1
@Var @RT(13)RedoStartData @RT(0) @T @T @DERIVED 0 @T @T @DT @RT(26)tevRedoIdentSpeedEventData @RT(0) @T @T @UNKNOWN 0 @F
@F @F
@T
@BEG_Attrib
3 @RT(0) @RT(0) @RT(0)
@END_Attrib
1 4 @F @F @F @F

@END_Dcl

@END_Export

@BEG_Export

@BEG_Algo
@POSTUPDATE_ALGORITHM @RT(16)pUpdateMaxStatus @STRUCTURED_TEXT
@RT(0) @RT(28)sv_IdentMaxSpeedState.Status @RT(9)PU_Task_7 @F @F
@END_Algo

@BEG_Dcl
@RT(16)DclTreeContainer
0
@END_Dcl

@END_Export

@BEG_Export

@BEG_Algo
@POSTUPDATE_ALGORITHM @RT(14)pUpdateMinRedo @STRUCTURED_TEXT
@RT(0) @RT(27)sv_IdentMinSpeedState.bRedo @RT(9)PU_Task_7 @F @F
@END_Algo

@BEG_Dcl
@RT(16)DclTreeContainer
1
@Var @RT(13)RedoStartData @RT(0) @T @T @DERIVED 0 @T @T @DT @RT(26)tevRedoIdentSpeedEventData @RT(0) @T @T @UNKNOWN 0 @F
@F @F
@T
@BEG_Attrib
3 @RT(0) @RT(0) @RT(0)
@END_Attrib
1 4 @F @F @F @F

@END_Dcl

@END_Export

@BEG_Export

@BEG_Algo
@POSTUPDATE_ALGORITHM @RT(16)pUpdateMinStatus @STRUCTURED_TEXT
@RT(0) @RT(28)sv_IdentMinSpeedState.Status @RT(9)PU_Task_7 @F @F
@END_Algo

@BEG_Dcl
@RT(16)DclTreeContainer
0
@END_Dcl

@END_Export

@BEG_Body
@TL(15)
(**************************************** WARNING ********************************************
 *** The KEBA Kemro K2 System including software is not intended for safety control tasks! ***
 ***                       For further information see Comment tab!                        ***
 *********************************************************************************************)

IF sv_IdentState.bRedo THEN
    IF sv_OperationMode <> nSetup THEN
       SET_ALARM(erSetupModeRequiredForCalib);
       sv_IdentState.bRedo := FALSE;
       RETURN;
    END_IF;
    RedoStartData.pMovement := @sv_IdentState;
    SET_EVENT(evRedoIdentStart, RedoStartData);
END_IF;

@END_Body

@@@BEG_Comment@@@
@TL(11)
@h    ! WARNING !
@h    The Kemro K2 system (including software) only meets category B according to EN 954-1,
@h    thus it is not intended for usage in safety-relevant control applications in the field
@h    of personal safety (e.g. emergency stop).
@h    To implement potentially necessary safety-relevant control tasks, always use additional
@h    external safety devices that are intended for the particular purpose, and meet the necessary
@h    functional safety.
@h    For further information see EN 954-1 (EN ISO 13849-1) and/or the K2-x00 user manual, chapter
@h    "CE conformity, directives and standards".

sets a evRedoStart event, which notifies the autocalibration FU to start this calibration movement
@@@END_Comment@@@

@BEG_Body
@TL(10)
(**************************************** WARNING ********************************************
 *** The KEBA Kemro K2 System including software is not intended for safety control tasks! ***
 ***                       For further information see Comment tab!                        ***
 *********************************************************************************************)

(* reset bRedo flag, when calibration is finished or aborted *)
IF sv_IdentState.Status <> tnCalibState_Running AND sv_IdentState.bRedo THEN
    sv_IdentState.bRedo := FALSE;
END_IF;

@END_Body

@@@BEG_Comment@@@
@TL(11)
@h    ! WARNING !
@h    The Kemro K2 system (including software) only meets category B according to EN 954-1,
@h    thus it is not intended for usage in safety-relevant control applications in the field
@h    of personal safety (e.g. emergency stop).
@h    To implement potentially necessary safety-relevant control tasks, always use additional
@h    external safety devices that are intended for the particular purpose, and meet the necessary
@h    functional safety.
@h    For further information see EN 954-1 (EN ISO 13849-1) and/or the K2-x00 user manual, chapter
@h    "CE conformity, directives and standards".

sets a evRedoStart event, which notifies the autocalibration FU to start this calibration movement
@@@END_Comment@@@

@BEG_Body
@TL(15)
(**************************************** WARNING ********************************************
 *** The KEBA Kemro K2 System including software is not intended for safety control tasks! ***
 ***                       For further information see Comment tab!                        ***
 *********************************************************************************************)

IF sv_IdentMaxSpeedState.bRedo THEN
    IF sv_OperationMode <> nSetup THEN
       SET_ALARM(erSetupModeRequiredForCalib);
       sv_IdentMaxSpeedState.bRedo := FALSE;
       RETURN;
    END_IF;
    RedoStartData.pMovement := @sv_IdentMaxSpeedState;
    SET_EVENT(evRedoIdentMaxSpeedStart, RedoStartData);
END_IF;

@END_Body

@@@BEG_Comment@@@
@TL(11)
@h    ! WARNING !
@h    The Kemro K2 system (including software) only meets category B according to EN 954-1,
@h    thus it is not intended for usage in safety-relevant control applications in the field
@h    of personal safety (e.g. emergency stop).
@h    To implement potentially necessary safety-relevant control tasks, always use additional
@h    external safety devices that are intended for the particular purpose, and meet the necessary
@h    functional safety.
@h    For further information see EN 954-1 (EN ISO 13849-1) and/or the K2-x00 user manual, chapter
@h    "CE conformity, directives and standards".

sets a evRedoStart event, which notifies the autocalibration FU to start this calibration movement
@@@END_Comment@@@

@BEG_Body
@TL(10)
(**************************************** WARNING ********************************************
 *** The KEBA Kemro K2 System including software is not intended for safety control tasks! ***
 ***                       For further information see Comment tab!                        ***
 *********************************************************************************************)

(* reset bRedo flag, when calibration is finished or aborted *)
IF sv_IdentMaxSpeedState.Status <> tnCalibState_Running AND sv_IdentMaxSpeedState.bRedo THEN
    sv_IdentMaxSpeedState.bRedo := FALSE;
END_IF;

@END_Body

@@@BEG_Comment@@@
@TL(11)
@h    ! WARNING !
@h    The Kemro K2 system (including software) only meets category B according to EN 954-1,
@h    thus it is not intended for usage in safety-relevant control applications in the field
@h    of personal safety (e.g. emergency stop).
@h    To implement potentially necessary safety-relevant control tasks, always use additional
@h    external safety devices that are intended for the particular purpose, and meet the necessary
@h    functional safety.
@h    For further information see EN 954-1 (EN ISO 13849-1) and/or the K2-x00 user manual, chapter
@h    "CE conformity, directives and standards".

sets a evRedoStart event, which notifies the autocalibration FU to start this calibration movement
@@@END_Comment@@@

@BEG_Body
@TL(15)
(**************************************** WARNING ********************************************
 *** The KEBA Kemro K2 System including software is not intended for safety control tasks! ***
 ***                       For further information see Comment tab!                        ***
 *********************************************************************************************)

IF sv_IdentMinSpeedState.bRedo THEN
    IF sv_OperationMode <> nSetup THEN
       SET_ALARM(erSetupModeRequiredForCalib);
       sv_IdentMinSpeedState.bRedo := FALSE;
       RETURN;
    END_IF;
    RedoStartData.pMovement := @sv_IdentMinSpeedState;
    SET_EVENT(evRedoIdentMinSpeedStart, RedoStartData);
END_IF;

@END_Body

@@@BEG_Comment@@@
@TL(11)
@h    ! WARNING !
@h    The Kemro K2 system (including software) only meets category B according to EN 954-1,
@h    thus it is not intended for usage in safety-relevant control applications in the field
@h    of personal safety (e.g. emergency stop).
@h    To implement potentially necessary safety-relevant control tasks, always use additional
@h    external safety devices that are intended for the particular purpose, and meet the necessary
@h    functional safety.
@h    For further information see EN 954-1 (EN ISO 13849-1) and/or the K2-x00 user manual, chapter
@h    "CE conformity, directives and standards".

sets a evRedoStart event, which notifies the autocalibration FU to start this calibration movement
@@@END_Comment@@@

@BEG_Body
@TL(10)
(**************************************** WARNING ********************************************
 *** The KEBA Kemro K2 System including software is not intended for safety control tasks! ***
 ***                       For further information see Comment tab!                        ***
 *********************************************************************************************)

(* reset bRedo flag, when calibration is finished or aborted *)
IF sv_IdentMinSpeedState.Status <> tnCalibState_Running AND sv_IdentMinSpeedState.bRedo THEN
    sv_IdentMinSpeedState.bRedo := FALSE;
END_IF;

@END_Body

@@@BEG_Comment@@@
@TL(11)
@h    ! WARNING !
@h    The Kemro K2 system (including software) only meets category B according to EN 954-1,
@h    thus it is not intended for usage in safety-relevant control applications in the field
@h    of personal safety (e.g. emergency stop).
@h    To implement potentially necessary safety-relevant control tasks, always use additional
@h    external safety devices that are intended for the particular purpose, and meet the necessary
@h    functional safety.
@h    For further information see EN 954-1 (EN ISO 13849-1) and/or the K2-x00 user manual, chapter
@h    "CE conformity, directives and standards".

sets a evRedoStart event, which notifies the autocalibration FU to start this calibration movement
@@@END_Comment@@@
@END_Body

@END_Contents
